// TIA Portal V18 export
TYPE "RCS_KeyenceSR1000_Output"
   STRUCT
      LatchAndErrorClearControl : Struct
         ReservedBit0 : Bool;
         ResultDataLatch : Bool;
         ReservedBit2 : Bool;
         ReservedBit3 : Bool;
         ReservedBit4 : Bool;
         ReservedBit5 : Bool;
         ReservedBit6 : Bool;
         ErrorClear : Bool;
      END_STRUCT;
      OperationInstructionControl : Struct
         ReadRequest : Bool;   // Reading start request
         PresetRequest : Bool;   // Preset reading start
         RegisterPresetDataRequest : Bool;
         TuneRequest : Bool;
         BloadRequest : Bool;
         ReservedBit5 : Bool;
         ReservedBit6 : Bool;
         ReservedBit7 : Bool;
      END_STRUCT;
      CompletionClearControl : Struct
         ReadCompleteClear : Bool;
         PresetCompleteClear : Bool;
         RegisterPresetDataCompleteClear : Bool;
         TuneCompleteClear : Bool;
         BloadCompleteClear : Bool;
         ReservedBit5 : Bool;
         ReservedBit6 : Bool;
         EXTRequestCompleteClear : Bool;
      END_STRUCT;
      ParameterBankNumber : Struct
         BankNo_BloadFileNo : UInt;
      END_STRUCT;
      UserData : Struct
         UserDataSize : UInt;
         UserData : Array[1..128] of Char;
      END_STRUCT;
   END_STRUCT;
END_TYPE
